TYPE "TAx_Speed_Ctrl"
VERSION : 0.1
// Block: TAx_Speed_Ctrl
   STRUCT
      SafeStop : Bool;
      Rst : Bool;
      RstHW : Bool;
      Power : Bool;
      MovePlus : Bool;
      MoveMinus : Bool;
      ExtControl : Bool;
      Velocity : LReal;
      Acceleration : LReal;
      Deceleration : LReal;
      Jerk : LReal;
   END_STRUCT;

END_TYPE
